{attribute 'qualified_only'}
VAR_GLOBAL
		EtherCAT_Master_APSxxxx : EtherCAT_Master_APSxxxx_C0802AAD;
END_VAR

(* stored: Version 1.2.0.0, ProductVersion 3.1.4024.9
   GVL GVL_iXlinker: Id {9e7cbec0-3e54-412a-bb50-f1e2ec3f0300} *)
